Universal Robots PolyScope program: DMT08b_9.urp

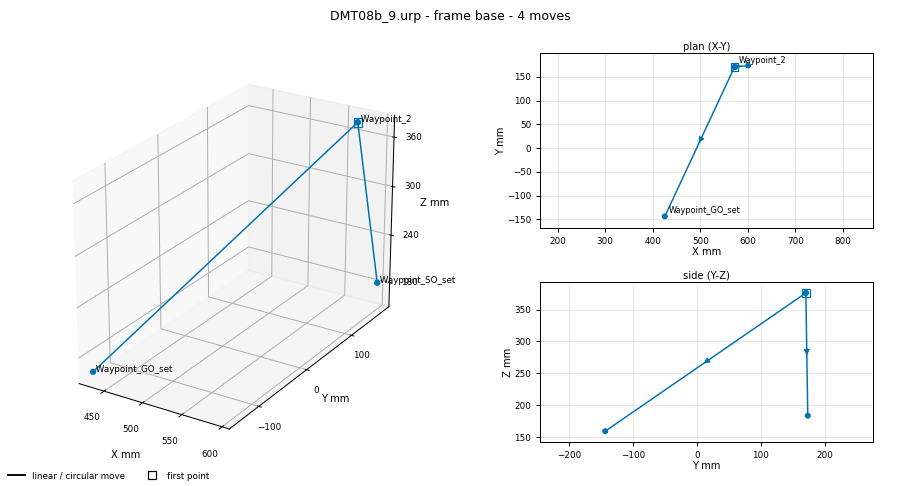
[picture p0: tool path of DMT08b_9.urp in frame base, 4 of 12 moves have a stored position in this frame; points joined in program order, loops and branches not executed]
Program DMT08b_9 (installation=default directory=/programs/usbdisk/DMT createdIn=3.5.0.10584 lastSavedIn=3.15.8.106339 robotSerialNumber=2017307354)
Calibrated DH parameters: a=[-0.000055, -0.610354, -0.571266, 0.000097, 0.000056, 0]; d=[0.128196, 3.8936, -4.338276, 0.608123, 0.115639, 0.092138]; alpha=[1.57086, -0.013529, -0.012604, 1.570975, -1.570813, 0]; deltaTheta=[-0.000051, -0.086091, 0.095923, -0.009846, -0.000078, 0.000069]
BeforeStart
  Script: enable_external_ft_sensor( True , sensor_mass = 0.0,  sensor_measuring_offset = [0.0, 0.0, 0.0], sensor_cog = [0.0, 0.0, 0.0] )
  sock_res := True
  Loop While (checkContinuously=false) expression=not sock_res
    Script: sock_res=socket_open("192.168.1.30",1000)
  res := ""
  Loop While (checkContinuously=false) expression=res ≟ ""
    Script: socket_send_line("TARE(1)")
    Script: res=socket_read_string()
  Script: write_output_boolean_register(0, False)
  Wait Sleep waitTime=0.01
  Script: popup("Registers reset, run PC code and then click Continue", title="Hi DMT", blocking = True)
  mode := 0
Robot Program (runOnlyOnce=true)
  Script: write_output_boolean_register(0, True)
  Script: sync()
  Loop While (checkContinuously=false) expression=mode<4
    MoveL speed 250 mm/s, acceleration 1200 mm/s^2 (useActiveTCP=true) feature=Base
      Waypoint Waypoint_2: TCP in base x=571.904 y=170.6 z=376.04 mm, rx=-3.0672 ry=-0.6069 rz=0.1286 rad; joints [180.011, -93.878, 121.325, -112.689, 269.302, 248.088] deg
    Loop While (checkContinuously=true) expression=mode==1
      Script: write_output_boolean_register(0, True)
      Script: sync()
      MoveL speed 250 mm/s, acceleration 1200 mm/s^2 (useActiveTCP=true) feature=Base
        Waypoint Waypoint_GO_set: TCP in base x=425.345 y=-143.617 z=159.528 mm, rx=-3.1406 ry=-0.0004 rz=-0.0004 rad; joints [139.43, -89.319, 148.344, -149.002, 269.754, 229.55] deg
      Force Simple feature=Base; selection=[0, 0, 1, 0, 0, 0]; wrench=[0, 0, -6, 0, 0, 0]; limitsForce=[0.15, 0.15, 0.15, 1.047198, 1.047198, 1.047198]; limitsMotion=[0.1, 0.1, 0.1, 0.349066, 0.349066, 0.349066]
        Wait Sleep waitTime=1
        MoveL speed 250 mm/s, acceleration 1200 mm/s^2 (useActiveTCP=true) feature=Base
          Waypoint Waypoint_3 (Relative): relativeFromPosition TCP in base x=425.349 y=-143.636 z=159.524 mm, rx=-3.1406 ry=-0.0004 rz=-0.0004 rad; joints [139.429, -89.317, 148.343, -149, 269.752, 229.546] deg; TCP in base x=345.34 y=-143.623 z=159.513 mm, rx=-3.1405 ry=-0.0007 rz=-0.0003 rad; joints [130.967, -97.907, 155.766, -147.823, 269.851, 221.067] deg
      Loop Counting (count=4) loopVariable(name=Loop_8)
        MoveL speed 250 mm/s, acceleration 1200 mm/s^2 (useActiveTCP=true) feature=Base
          Waypoint Waypoint_1 (Relative): relativeFromPosition TCP in base x=420.336 y=-78.634 z=159.533 mm, rx=-3.1406 ry=-0.0007 rz=-0.0003 rad; joints [146.377, -91.505, 150.482, -148.956, 269.78, 236.483] deg; TCP in base x=420.31 y=-78.604 z=162.495 mm, rx=-3.1405 ry=-0.0008 rz=-0.0002 rad; joints [146.375, -91.989, 150.362, -148.346, 269.782, 236.481] deg
        MoveL speed 50 mm/s, acceleration 300 mm/s^2 (useActiveTCP=true) feature=Base
          Waypoint Waypoint_G23 (Relative): relativeFromPosition TCP in base x=345.312 y=-143.593 z=159.488 mm, rx=-3.1405 ry=-0.0007 rz=-0.0003 rad; joints [130.967, -97.908, 155.771, -147.824, 269.851, 221.065] deg; TCP in base x=420.327 y=-78.625 z=159.524 mm, rx=-3.1406 ry=-0.0007 rz=-0.0002 rad; joints [146.378, -91.505, 150.483, -148.954, 269.778, 236.483] deg
        MoveL speed 50 mm/s, acceleration 300 mm/s^2 (useActiveTCP=true) feature=Base
          Waypoint Waypoint_G4O (Relative): relativeFromPosition TCP in base x=409.862 y=-222.419 z=100.846 mm, rx=3.141 ry=0 rz=0 rad; joints [137.981, -73.268, 126.217, -142.972, 269.975, 227.981] deg; TCP in base x=409.862 y=-222.419 z=98.846 mm, rx=3.141 ry=0 rz=0 rad; joints [137.981, -73, 126.297, -143.319, 269.975, 227.981] deg
        Force Simple feature=Base; selection=[0, 0, 1, 0, 0, 0]; wrench=[0, 0, -1, 0, 0, 0]; limitsForce=[0.15, 0.15, 0.15, 1.047198, 1.047198, 1.047198]; limitsMotion=[0.1, 0.1, 0.1, 0.349066, 0.349066, 0.349066]
          Wait Sleep waitTime=1
          MoveL speed 250 mm/s, acceleration 1200 mm/s^2 (useActiveTCP=true) feature=Base
            Waypoint Waypoint_3 (Relative): relativeFromPosition TCP in base x=425.349 y=-143.636 z=159.524 mm, rx=-3.1406 ry=-0.0004 rz=-0.0004 rad; joints [139.429, -89.317, 148.343, -149, 269.752, 229.546] deg; TCP in base x=345.34 y=-143.623 z=159.513 mm, rx=-3.1405 ry=-0.0007 rz=-0.0003 rad; joints [130.967, -97.907, 155.766, -147.823, 269.851, 221.067] deg
      MoveL speed 250 mm/s, acceleration 1200 mm/s^2 (useActiveTCP=true) feature=Base
        Waypoint Waypoint_2: TCP in base x=571.904 y=170.6 z=376.04 mm, rx=-3.0672 ry=-0.6069 rz=0.1286 rad; joints [180.011, -93.878, 121.325, -112.689, 269.302, 248.088] deg
      Script: write_output_boolean_register(0, False)
      Script: sync()
    SuppressedNode
      Loop While (checkContinuously=true) expression=mode==2
        Script: write_output_boolean_register(0, True)
        Script: write_output_boolean_register(32, True)
        Script: sync()
        Wait Sleep waitTime=0.5
        MoveL speed 250 mm/s, acceleration 1200 mm/s^2 (useActiveTCP=true) feature=Base
          Waypoint Waypoint_DO_set: TCP in base x=932.962 y=-58.379 z=442.977 mm, rx=3.141 ry=0.0001 rz=0.0001 rad; joints [165.794, -65.483, 81.029, -105.558, 269.02, 256.304] deg
          Waypoint Waypoint_DO1 (Relative): relativeFromPosition TCP in base x=658.55 y=-49.546 z=529.242 mm, rx=3.1409 ry=0.0002 rz=0 rad; joints [166.189, -63.237, 41.872, -68.645, 269.959, 256.184] deg; TCP in base x=658.55 y=-49.546 z=499.242 mm, rx=3.1409 ry=0.0002 rz=0 rad; joints [166.189, -65.044, 49.207, -74.172, 269.959, 256.184] deg
        Script: write_output_boolean_register(32, False)
        Wait Sleep waitTime=1
        MoveL speed 250 mm/s, acceleration 1200 mm/s^2 (useActiveTCP=true) feature=Base
          Waypoint Waypoint_D1O (Relative): relativeFromPosition TCP in base x=658.55 y=-49.546 z=499.242 mm, rx=3.1409 ry=0.0002 rz=0 rad; joints [166.189, -65.044, 49.207, -74.172, 269.959, 256.184] deg; TCP in base x=658.55 y=-49.546 z=529.242 mm, rx=3.1409 ry=0.0002 rz=0 rad; joints [166.189, -63.237, 41.872, -68.645, 269.959, 256.184] deg
        Script: write_output_boolean_register(0, False)
        Script: sync()
    Loop While (checkContinuously=true) expression=mode==3
      Script: write_output_boolean_register(0, True)
      Script: write_output_boolean_register(32, True)
      MoveL speed 100 mm/s, acceleration 200 mm/s^2 (useActiveTCP=false) feature=Base
        Waypoint Waypoint_SO_set: motionParameters(nextMotionTime=2); TCP in base x=600.623 y=173.61 z=183.794 mm, rx=-3.0823 ry=-0.6058 rz=-0.0104 rad; joints [180.371, -77.146, 129.397, -142.624, 269.551, 248.303] deg
      Script: sync()
      MoveL speed 100 mm/s, acceleration 200 mm/s^2 (useActiveTCP=true) feature=Base
        Waypoint Waypoint_SO1 (Relative): motionParameters(nextMotionTime=1.5); relativeFromPosition TCP in base x=600.643 y=173.605 z=183.787 mm, rx=-3.0823 ry=-0.6058 rz=-0.0104 rad; joints [180.371, -77.144, 129.395, -142.626, 269.552, 248.303] deg; TCP in base x=685.651 y=173.612 z=183.778 mm, rx=-3.0824 ry=-0.6061 rz=-0.0104 rad; joints [180.262, -71.012, 120.459, -139.819, 269.436, 248.192] deg
      SuppressedNode
        Script: write_output_boolean_register(32, True)
      SuppressedNode
        Script: sync()
      MoveL speed 100 mm/s, acceleration 200 mm/s^2 (useActiveTCP=true) feature=Base
        Waypoint Waypoint_S12 (Relative): relativeFromPosition TCP in base x=685.629 y=173.589 z=183.77 mm, rx=-3.0824 ry=-0.606 rz=-0.0103 rad; joints [180.26, -71.013, 120.461, -139.819, 269.438, 248.193] deg; TCP in base x=786.108 y=171.091 z=164.679 mm, rx=-3.0833 ry=-0.6014 rz=-0.0106 rad; joints [179.995, -62.654, 109.746, -137.472, 269.306, 248.083] deg
      Wait Sleep waitTime=0.5
      SuppressedNode
        Script: write_output_boolean_register(32, False)
      SuppressedNode
        Script: sync()
      SuppressedNode
        Script: write_output_boolean_register(32, True)
      SuppressedNode
        Script: sync()
      SuppressedNode
        Force Simple feature=Base; selection=[0, 0, 1, 0, 0, 0]; wrench=[0, 0, -6, 0, 0, 0]; limitsForce=[0.15, 0.15, 0.15, 1.047198, 1.047198, 1.047198]; limitsMotion=[0.1, 0.1, 0.1, 0.349066, 0.349066, 0.349066]
          Placeholder
      Script: write_output_boolean_register(32, False)
      Script: sync()
      MoveL speed 30 mm/s, acceleration 200 mm/s^2 (useActiveTCP=false) feature=Base
        Waypoint Waypoint_S23 (Relative): relativeFromPosition TCP in base x=785.648 y=173.445 z=163.163 mm, rx=-3.0824 ry=-0.606 rz=-0.0107 rad; joints [180.167, -62.54, 109.774, -137.619, 269.309, 248.082] deg; TCP in base x=710.561 y=173.464 z=163.11 mm, rx=-3.0823 ry=-0.6063 rz=-0.0105 rad; joints [180.231, -67.597, 118.273, -141.052, 269.407, 248.131] deg
      Script: write_output_boolean_register(0, False)
      Script: sync()
    Loop While (checkContinuously=true) expression=mode==4
      Halt
  Script: sync()
Thread Thread_1 (runOnlyOnce=false)
  tmp := p[0,0,0,0,0,0]
  Loop Forever
    Script file /home/ur/ursim/ursim-3.15.0.106151/programs/pose_register.script
      | tmp[0]=read_input_float_register(0)
      | tmp[1]=read_input_float_register(1)
      | tmp[2]=read_input_float_register(2)
      | tmp[3]=read_input_float_register(3)
      | tmp[4]=read_input_float_register(4)
      | tmp[5]=read_input_float_register(5)
    Script: sync()
    mode := read_input_integer_register(0)
    Script: sync()
